(* CODESYS project VERSENY_25_F2

Project tree, tasks and I/O mapping:
  Device : CODESYS Control for PFC200 SL, 3S - Smart Software Solutions GmbH, version 4.1.0.0
    application Application
      libraries: Standard, 3.5.18.0 (System)
      task MainTask (cyclic, interval t#20ms, priority 1) calls PRG_TRIG, TESTPRG
      function BETWEEN [ST]
      CIMKEZO/
        data type ENUCIMKEZO
        function block FBCIMKEZO [ST]
      DOBOZ/
        data type ENUDOBOZ
        function block FBDOBOZ [ST]
      function block FBDOBOZ21212 [ST]
      global variables GVL
      global variables I
      LIFT/
        data type ENULIFT
        function block FBLIFT [ST]
      PALETTAZO/
        data type ENUPALETTAZO
        function block FBPALETTAZO [ST]
      program PLC_PRG [ST]
      PRESET/
        data type ENUPRESET
        function block FBPRESET [ST]
      program PRG_TRIG [ST]
      global variables Q
      RAKLAP/
        data type ENURAKLAP
        function block FBRAKLAP [ST]
      data type STATE
      program TESTPRG [ST]
      function block VILLOGO4 [ST]
    Pfc200Bus : Wago PFC200 internal bus, 3S - Smart Software Solutions GmbH, version 4.1.0.0
      _750_14xx_1 : 16DI, WAGO Kontakttechnik GmbH u. Co. KG, order no. 750-14xx, version 4.1.0.0
          unmapped channels: %IW10 Digital Inputs 0 - 15
      _750_14xx : 16DI, WAGO Kontakttechnik GmbH u. Co. KG, order no. 750-14xx, version 4.1.0.0
          unmapped channels: %IW5 Digital Inputs 0 - 15
      _750_15xx_1 : 16DO, WAGO Kontakttechnik GmbH u. Co. KG, order no. 750-15xx, version 4.1.0.0
          unmapped channels: %QW10 Digital Outputs 0 - 15
      _750_15xx : 16DO, WAGO Kontakttechnik GmbH u. Co. KG, order no. 750-15xx, version 4.1.0.0
          unmapped channels: %QW5 Digital Outputs 0 - 15
      _75x_459 : 75x-459/0..-000 4AI, 0-10 V, WAGO Kontakttechnik GmbH u. Co. KG, order no. 75x-459(/0..-000), version 4.1.0.0
          unmapped channels: Analog Input Channel 0, Analog Input Channel 1, Analog Input Channel 2, Analog Input Channel 3
      _75x_559 : 75x-559/0..-000 4AO, 0-10 V, WAGO Kontakttechnik GmbH u. Co. KG, order no. 75x-559(/0..-000), version 4.1.0.0
          unmapped channels: Analog Output Channel 0, Analog Output Channel 1, Analog Output Channel 2, Analog Output Channel 3
*)

// Device/Application/STATE
{attribute 'qualified_only'}
{attribute 'strict'}
TYPE STATE :
(
	enum_member := 0
);
END_TYPE

// Device/Application/CIMKEZO/ENUCIMKEZO
{attribute 'qualified_only'}
//{attribute 'strict'}
TYPE ENUCIMKEZO:
(
	PRESET := 0,
	CIMKEZZ := 1,
	DONE := 2
);
END_TYPE

// Device/Application/DOBOZ/ENUDOBOZ
{attribute 'qualified_only'}
//{attribute 'strict'}
TYPE ENUDOBOZ:
(
	PRESET := 0,
	CIKMEZO_CLEAR := 1,
	DONE := 2,
	GO := 3
);
END_TYPE

// Device/Application/LIFT/ENULIFT
{attribute 'qualified_only'}
//{attribute 'strict'}
TYPE ENULIFT:
(
	PRESET := 0,
	PARANCS_FEL := 1,
	PARANCS_LE := 2,
	LIFT_MOZOG := 3,
	DONE := 4
);
END_TYPE

// Device/Application/PALETTAZO/ENUPALETTAZO
{attribute 'qualified_only'}
//{attribute 'strict'}
TYPE ENUPALETTAZO:
(
	PRESET := 0,
	ELHALADT := 1,
	CELBA_ERT := 2,
	DOBOZOK_KESZ := 3,
	PALETTAZORA_TOVABBIT := 4,
	MEGERKEZETT := 5,
	BETOLO_VISSZA := 6,
	BETOLO_MEGY := 7,
	BETOLO_KESZ := 8,
	MEGFOG := 9,
	KINYIT := 10,
	DONE := 11
);
END_TYPE

// Device/Application/PRESET/ENUPRESET

{attribute 'qualified_only'}
//{attribute 'strict'}
TYPE ENUPRESET:
(
	PRESET := 0,
	MINDEN_LELAITAS := 1,
	LIFT_VISSZA := 2,
	DONE := 3
);
END_TYPE

// Device/Application/RAKLAP/ENURAKLAP
{attribute 'qualified_only'}
//{attribute 'strict'}
TYPE ENURAKLAP:
(
	PRESET := 0,
	WAIT := 1,
	DONE := 2,
	LEFELE := 3,
	LIFT_LE_VEGALAS := 4,
	LIFTBOL_KI := 5,
	LIFTBOL_KI_KETO := 6,
	GORGOS_MEHET := 7,
	BERAKO_INDIT := 8,
	LIFT_BEHORDO := 9,
	LIFT_FEL := 10,
	FELADAT_DONE := 11
);
END_TYPE

// Device/Application/GVL
{attribute 'qualified_only'}
VAR_GLOBAL
	STATE : STATE;
END_VAR

// Device/Application/I
{attribute 'qualified_only'}
VAR_GLOBAL
END_VAR

// Device/Application/Q
{attribute 'qualified_only'}
VAR_GLOBAL
END_VAR

// Device/Application/PRG_TRIG
PROGRAM PRG_TRIG
VAR
END_VAR

END_PROGRAM

// Device/Application/TESTPRG
PROGRAM TESTPRG
VAR
	LIFT : FBLIFT;
	FELFELE : BOOL;
	LEFELE : BOOL;
END_VAR

//LIFT TESZTELESE
IF I.I0 THEN
	FELFELE := TRUE;
	LEFELE := FALSE;
ELSIF I.I1 THEN
	LEFELE := TRUE;
	FELFELE := FALSE;
END_IF

LIFT(
	LEFELE:= LEFELE, 
	FELFELE:= FELFELE, 
	VEGALLASIG:= I.I2, 
	EN:= (I.I0 XOR I.I1), 
	DONE=> Q.Q0);

END_PROGRAM

// Device/Application/LIFT/FBLIFT
FUNCTION_BLOCK FBLIFT
VAR_INPUT
	LEFELE: BOOL;
	FELFELE: BOOL;
	VEGALLASIG: BOOL;
	EN: BOOL;
END_VAR
VAR_OUTPUT
	DONE: BOOL := FALSE;
END_VAR
VAR_IN_OUT
END_VAR
VAR
	LIFT: ENULIFT := ENULIFT.PRESET;
	VILLOGO4_PARANCS_VEGALLASIG_1_Q1: BOOL;
	BLANK_PARANCS_VEGALLASIG_1: BOOL;
	VILLOGO4_PARANCS_VEGALLASIG_1: VILLOGO4;
	TRANS_PARANCS_VEGALLASIG_PARANCS_FEL_T: TON;
	LELFELE: BOOL;
	TRANS_PARANCS_VEGALLASIG_PARANCS_LE_T: TON;
END_VAR

VILLOGO4_PARANCS_VEGALLASIG_1(T1:= T#1S, T2:= T#1S, T3:= T#0S, T4:= T#0S, Q1:= VILLOGO4_PARANCS_VEGALLASIG_1_Q1, Q2:= BLANK_PARANCS_VEGALLASIG_1, Q3:= BLANK_PARANCS_VEGALLASIG_1, Q4:= BLANK_PARANCS_VEGALLASIG_1, EN:= (LIFT = ENULIFT.PARANCS_VEGALLASIG));
TRANS_PARANCS_VEGALLASIG_PARANCS_FEL_T(PT:= T#5S, IN:= FELFELE AND (LIFT = ENULIFT.PARANCS_VEGALLASIG));
TRANS_PARANCS_VEGALLASIG_PARANCS_LE_T(PT:= T#5S, IN:= LELFELE AND (LIFT = ENULIFT.PARANCS_VEGALLASIG));

IF NOT EN THEN
	LIFT := ENULIFT.PRESET;
	LELFELE := FALSE;
	BLANK_PARANCS_VEGALLASIG_1 := FALSE;
	VILLOGO4_PARANCS_VEGALLASIG_1_Q1 := FALSE;
	DONE := FALSE;
	RETURN;
END_IF


CASE LIFT OF
	ENULIFT.PRESET:
	Q.LIFT_VEGALLASIG := VEGALLASIG;

	IF FELFELE AND NOT VEGALLASIG THEN
		LIFT := ENULIFT.PARANCS_FEL;
	ELSIF LEFELE AND NOT VEGALLASIG THEN
		LIFT := ENULIFT.PARANCS_LE;
	ELSIF VEGALLASIG AND (FELFELE OR LEFELE) THEN
		LIFT := ENULIFT.PARANCS_VEGALLASIG;
	END_IF

	ENULIFT.PARANCS_FEL:
	Q.LIFT_FEL := TRUE;

	IF I.LIFT_MOZOG THEN
		LIFT := ENULIFT.LIFT_MOZOG;
	END_IF

	ENULIFT.PARANCS_LE:
	Q.LIFT_LE := TRUE;

	IF I.LIFT_MOZOG THEN
		LIFT := ENULIFT.LIFT_MOZOG;
	END_IF


	ENULIFT.LIFT_MOZOG:
	IF NOT (VEGALLASIG AND NOT I.I15) THEN
		Q.LIFT_FEL := FALSE;
		Q.LIFT_LE := FALSE;
		Q.LIFT_VEGALLASIG := FALSE;
	END_IF

	IF GVL.LIFT_MOZOG_F_TRIG.Q THEN
		Q.LIFT_FEL := FALSE;
		Q.LIFT_LE := FALSE;
		Q.LIFT_VEGALLASIG := FALSE;
		

		LIFT := ENULIFT.DONE;
	END_IF



	ENULIFT.PARANCS_VEGALLASIG:

	IF TRANS_PARANCS_VEGALLASIG_PARANCS_FEL_T.Q THEN
		LIFT := ENULIFT.PARANCS_FEL;
	ELSIF TRANS_PARANCS_VEGALLASIG_PARANCS_LE_T.Q THEN
		LIFT := ENULIFT.PARANCS_LE;
	END_IF

END_CASE

DONE := (LIFT = ENULIFT.DONE);
Q.HORN := (VILLOGO4_PARANCS_VEGALLASIG_1_Q1 AND (LIFT = ENULIFT.PARANCS_VEGALLASIG));

END_FUNCTION_BLOCK

// Device/Application/VILLOGO4
FUNCTION_BLOCK VILLOGO4
VAR_INPUT
	T1: TIME;
	T2: TIME;
	T3: TIME;
	T4: TIME;
END_VAR
VAR_IN_OUT
	Q1: BOOL;
	Q2: BOOL;
	Q3: BOOL;
	Q4: BOOL;
END_VAR
VAR
	T1_TON: TON;
	T2_TON: TON;
	T3_TON: TON;
	T4_TON: TON;
END_VAR
VAR_INPUT
	EN: BOOL := FALSE;
END_VAR
VAR
	EN_F_TRIG: F_TRIG;
	EN_R_TRIG: R_TRIG;
	STATE: INT := 0;
	PREV_STATE: INT := 0;
END_VAR

EN_F_TRIG(CLK := EN);
EN_R_TRIG(CLK := EN);

IF EN_F_TRIG.Q THEN
	Q1 := FALSE;
	Q2 := FALSE;
	Q3 := FALSE;
	Q4 := FALSE;
	T1_TON.PT := T1_TON.ET;
	T2_TON.PT := T2_TON.ET;
	T3_TON.PT := T3_TON.ET;
	T4_TON.PT := T4_TON.ET;
	STATE := 0;
ELSIF EN_R_TRIG.Q THEN
		Q1 := TRUE;
END_IF

IF NOT EN THEN
	RETURN;
END_IF

T1_TON(IN:= EN_R_TRIG.Q OR (STATE = 0), PT:= T1);
T2_TON(IN:= STATE = 1, PT:= T2);
T3_TON(IN:= STATE = 2, PT:= T3);
T4_TON(IN:= STATE = 3, PT:= T4);

IF T1_TON.Q THEN
	Q1 := FALSE;
	Q2 := TRUE;
END_IF
IF T2_TON.Q THEN
	Q2 := FALSE;
	Q3 := TRUE;
END_IF
IF T3_TON.Q THEN
	Q3 := FALSE;
	Q4 := TRUE;
END_IF
IF T4_TON.Q THEN
	Q4 := FALSE;
	Q1 := TRUE;
END_IF

IF T1_TON.Q OR T2_TON.Q OR T3_TON.Q OR T4_TON.Q THEN
	STATE := STATE + 1;
END_IF

IF STATE > 3 THEN
	STATE := 0;
END_IF

END_FUNCTION_BLOCK

// Device/Application/BETWEEN
FUNCTION BETWEEN : BOOL
VAR_INPUT
	STATE : INT;
	LOW : INT;
	HIGH : INT;
END_VAR
VAR_OUTPUT
END_VAR
VAR
	EN_TRIG : F_TRIG;
END_VAR

IF STATE >= LOW AND STATE <= HIGH THEN
	BETWEEN := TRUE;
ELSE 
	BETWEEN := FALSE;
END_IF

END_FUNCTION

// Device/Application/FBDOBOZ21212
FUNCTION_BLOCK FBDOBOZ21212
VAR_INPUT
	EN : BOOL;
END_VAR
VAR_OUTPUT
	DONE : BOOL;
END_VAR
VAR
END_VAR

END_FUNCTION_BLOCK

// Device/Application/PLC_PRG
PROGRAM PLC_PRG
VAR
END_VAR

%QW10 := %IW10;

END_PROGRAM

// Device/Application/CIMKEZO/FBCIMKEZO
FUNCTION_BLOCK FBCIMKEZO
VAR_INPUT
	EN: BOOL;
END_VAR
VAR_OUTPUT
	DONE: BOOL := FALSE;
END_VAR
VAR_IN_OUT
END_VAR
VAR
	CIMKEZO: ENUCIMKEZO := ENUCIMKEZO.PRESET;
	TRANS_CIMKEZZ_DONE_T: TON;
END_VAR

TRANS_CIMKEZZ_DONE_T(PT:= GVL.CIMKEZO_TIME, IN:= (CIMKEZO = ENUCIMKEZO.CIMKEZZ));

IF NOT EN THEN
	CIMKEZO := ENUCIMKEZO.PRESET;
	DONE := FALSE;
	RETURN;
END_IF


CASE CIMKEZO OF

	ENUCIMKEZO.PRESET:

	IF GVL.DOBOZ_CIMKEZONEL_F_TRIG.Q THEN
		CIMKEZO := ENUCIMKEZO.CIMKEZZ;
	END_IF


	ENUCIMKEZO.CIMKEZZ:

	IF TRANS_CIMKEZZ_DONE_T.Q THEN
		CIMKEZO := ENUCIMKEZO.DONE;
	END_IF


	ENUCIMKEZO.DONE:

	IF TRUE THEN
		CIMKEZO := ENUCIMKEZO.PRESET;
	END_IF

END_CASE

DONE := (CIMKEZO = ENUCIMKEZO.DONE);
Q.CIMKEZO := (CIMKEZO = ENUCIMKEZO.CIMKEZZ);

END_FUNCTION_BLOCK

// Device/Application/DOBOZ/FBDOBOZ
FUNCTION_BLOCK FBDOBOZ
VAR_INPUT
	MODE: BOOL;
	EN: BOOL;
END_VAR
VAR_OUTPUT
	DONE: BOOL := FALSE;
END_VAR
VAR_IN_OUT
END_VAR
VAR
	DOBOZ: ENUDOBOZ := ENUDOBOZ.PRESET;
	CIMKEZO: FBCIMKEZO;
	PALETTAZO: FBPALETTAZO;
	MAX_DOBOZ: INT;
	MAX_OSZLOP: INT;
END_VAR

PALETTAZO(MAX_DOBOZ := MAX_DOBOZ, MAX_OSZLOP := MAX_OSZLOP, EN:= (DOBOZ = ENUDOBOZ.CIKMEZO_CLEAR) OR (DOBOZ = ENUDOBOZ.GO));
CIMKEZO(EN:= (DOBOZ = ENUDOBOZ.GO));

IF NOT EN THEN
	DOBOZ := ENUDOBOZ.PRESET;
	MAX_OSZLOP := 0;
	MAX_DOBOZ := 0;
	DONE := FALSE;
	RETURN;
END_IF


CASE DOBOZ OF

	ENUDOBOZ.PRESET:

	IF TRUE THEN
		DOBOZ := ENUDOBOZ.GO;
	END_IF


	ENUDOBOZ.CIKMEZO_CLEAR:

	IF TRUE THEN
		DOBOZ := ENUDOBOZ.GO;
	END_IF



	ENUDOBOZ.GO:
	IF MODE THEN
		Q.TERELO := TRUE;
		MAX_DOBOZ := 3;
		MAX_OSZLOP := 2;
	ELSE
		Q.TERELO := FALSE;
		MAX_DOBOZ := 2;
		MAX_OSZLOP := 3;
	END_IF

	IF CIMKEZO.DONE THEN
		DOBOZ := ENUDOBOZ.CIKMEZO_CLEAR;
	ELSIF PALETTAZO.DONE THEN
		DOBOZ := ENUDOBOZ.DONE;
	END_IF

END_CASE

DONE := (DOBOZ = ENUDOBOZ.DONE);

END_FUNCTION_BLOCK

// Device/Application/PALETTAZO/FBPALETTAZO
FUNCTION_BLOCK FBPALETTAZO
VAR_INPUT
	MAX_DOBOZ: INT;
	MAX_OSZLOP: INT;
	EN: BOOL;
END_VAR
VAR_OUTPUT
	ATHALADT_DOBOZOK: INT;
	KESZ_OSZLOPOK: INT;
	DONE: BOOL := FALSE;
END_VAR
VAR_IN_OUT
END_VAR
VAR
	PALETTAZO: ENUPALETTAZO := ENUPALETTAZO.PRESET;
	TRANS_ELHALADT_CELBA_ERT_T: TON;
	ATHALADT_DOBOZOK_SZAMA: INT;
END_VAR

TRANS_ELHALADT_CELBA_ERT_T(PT:= GVL.CELBA_ER_TIME, IN:= (PALETTAZO = ENUPALETTAZO.ELHALADT));

IF NOT EN THEN
	PALETTAZO := ENUPALETTAZO.PRESET;
	ATHALADT_DOBOZOK_SZAMA := 0;
	DONE := FALSE;
	KESZ_OSZLOPOK := 0;
	ATHALADT_DOBOZOK := 0;
	RETURN;
END_IF


CASE PALETTAZO OF
	ENUPALETTAZO.PRESET:
	Q.BEHORDO := TRUE;
	Q.PALETTAZO_OPEN := FALSE;

	IF GVL.BEHORDO_Z1_R_TRIG.Q THEN
		PALETTAZO := ENUPALETTAZO.MEGERKEZETT;
	END_IF


	ENUPALETTAZO.ELHALADT:

	IF TRANS_ELHALADT_CELBA_ERT_T.Q THEN
		ATHALADT_DOBOZOK_SZAMA := ATHALADT_DOBOZOK_SZAMA + 1;

		PALETTAZO := ENUPALETTAZO.CELBA_ERT;
	END_IF


	ENUPALETTAZO.CELBA_ERT:

	IF ATHALADT_DOBOZOK_SZAMA < MAX_DOBOZ THEN
		PALETTAZO := ENUPALETTAZO.PRESET;
	ELSIF ATHALADT_DOBOZOK_SZAMA = MAX_DOBOZ THEN
		PALETTAZO := ENUPALETTAZO.DOBOZOK_KESZ;
	END_IF

	ENUPALETTAZO.DOBOZOK_KESZ:
	Q.BEHORDO := FALSE;
	Q.PALETTAZO_SZALAG := FALSE;

	IF I.PALETTAZO_CLOSED AND I.PALETTAZO_BETOLO_VEGALLAS AND I.PALETTAZO_DOBOZ_MEGFOGVA AND NOT Q.PALETTAZO_BETOLO AND NOT Q.PALETTAZO_MEGFOGO THEN
		PALETTAZO := ENUPALETTAZO.PALETTAZORA_TOVABBIT;
	END_IF


	ENUPALETTAZO.PALETTAZORA_TOVABBIT:

	IF GVL.PALETTAZO_BETOLO_VEGALLAS_R_TRIG.Q THEN
		PALETTAZO := ENUPALETTAZO.BETOLO_VISSZA;
	END_IF

	ENUPALETTAZO.MEGERKEZETT:
	Q.PALETTAZO_SZALAG := TRUE;

	IF GVL.BEHORDO_Z1_F_TRIG.Q THEN
		PALETTAZO := ENUPALETTAZO.ELHALADT;
	END_IF


	ENUPALETTAZO.BETOLO_VISSZA:

	IF GVL.PALETTAZO_BETOLO_VEGALLAS_F_TRIG.Q THEN
		PALETTAZO := ENUPALETTAZO.BETOLO_MEGY;
	END_IF


	ENUPALETTAZO.BETOLO_MEGY:

	IF GVL.PALETTAZO_BETOLO_VEGALLAS_R_TRIG.Q THEN
		KESZ_OSZLOPOK := KESZ_OSZLOPOK + 1;

		PALETTAZO := ENUPALETTAZO.BETOLO_KESZ;
	END_IF


	ENUPALETTAZO.BETOLO_KESZ:

	IF KESZ_OSZLOPOK < MAX_OSZLOP THEN
		PALETTAZO := ENUPALETTAZO.PRESET;
	ELSIF KESZ_OSZLOPOK = MAX_OSZLOP THEN
		PALETTAZO := ENUPALETTAZO.MEGFOG;
	END_IF


	ENUPALETTAZO.MEGFOG:

	IF GVL.PALETTAZO_DOBOZ_MEGFOGVA_R_TRIG.Q AND NOT I.LIFT_MOZOG THEN
		PALETTAZO := ENUPALETTAZO.KINYIT;
	END_IF

	ENUPALETTAZO.KINYIT:
	Q.PALETTAZO_OPEN := TRUE;

	IF TRUE THEN
		PALETTAZO := ENUPALETTAZO.DONE;
	END_IF


END_CASE

DONE := (PALETTAZO = ENUPALETTAZO.DONE);
Q.PALETTAZO_BETOLO := (PALETTAZO = ENUPALETTAZO.PALETTAZORA_TOVABBIT);
Q.PALETTAZO_MEGFOGO := (PALETTAZO = ENUPALETTAZO.MEGFOG);

END_FUNCTION_BLOCK

// Device/Application/PRESET/FBPRESET
FUNCTION_BLOCK FBPRESET
VAR_INPUT
	EN: BOOL;
END_VAR
VAR_OUTPUT
	DONE: BOOL := FALSE;
END_VAR
VAR_IN_OUT
END_VAR
VAR
	PRESET: ENUPRESET := ENUPRESET.PRESET;
END_VAR

IF NOT EN THEN
	PRESET := ENUPRESET.PRESET;
	DONE := FALSE;
	RETURN;
END_IF


CASE PRESET OF

	ENUPRESET.PRESET:

	IF EN THEN
		PRESET := ENUPRESET.MINDEN_LELAITAS;
	END_IF


	ENUPRESET.MINDEN_LELAITAS:
	%QW10 := 0;

	IF TRUE THEN
		PRESET := ENUPRESET.LIFT_VISSZA;
	END_IF


	ENUPRESET.LIFT_VISSZA:

	IF GVL.LIFT_MOZOG_F_TRIG.Q OR GVL.LIFT_LENT THEN
		PRESET := ENUPRESET.DONE;
	END_IF


END_CASE

DONE := (PRESET = ENUPRESET.DONE);
Q.LIFT_LE := (PRESET = ENUPRESET.LIFT_VISSZA);

END_FUNCTION_BLOCK

// Device/Application/RAKLAP/FBRAKLAP
FUNCTION_BLOCK FBRAKLAP
VAR_INPUT
	LEFELE: BOOL;
	KIRAKAS: BOOL;
	BERAKAS: BOOL;
	HARMADIK: BOOL;
	STOP: BOOL;
	EN: BOOL;
END_VAR
VAR_OUTPUT
	FELADAT_DONE: BOOL;
	DONE: BOOL := FALSE;
END_VAR
VAR_IN_OUT
END_VAR
VAR
	RAKLAP: ENURAKLAP := ENURAKLAP.PRESET;
	LIFT: FBLIFT;
	LEFELE_MENJ: BOOL;
	FELFELE_MENJ: BOOL;
	VEGALAS_MENJ: BOOL;
	LIFT_BEHORDO: BOOL;
	TRANS_GORGOS_MEHET_DONE_T: TON;
	IDOMENTES : TIME;
END_VAR

LIFT(EN:= (RAKLAP = ENURAKLAP.LEFELE) OR 
		  (RAKLAP = ENURAKLAP.LIFT_FEL) OR 
          (RAKLAP = ENURAKLAP.LIFT_LE_VEGALAS) );
TRANS_GORGOS_MEHET_DONE_T(PT:= T#3S, IN:= ((RAKLAP = ENURAKLAP.GORGOS_MEHET) AND (NOT STOP)) );

LIFT.FELFELE := FELFELE_MENJ;
LIFT.LEFELE := LEFELE_MENJ;
LIFT.VEGALLASIG := VEGALAS_MENJ;


IF NOT EN THEN
	RAKLAP := ENURAKLAP.PRESET;
	LIFT_BEHORDO := FALSE;
	VEGALAS_MENJ := FALSE;
	FELFELE_MENJ := FALSE;
	LEFELE_MENJ := FALSE;
	DONE := FALSE;
	FELADAT_DONE := FALSE;
	RETURN;
END_IF


CASE RAKLAP OF

	ENURAKLAP.PRESET:

	IF EN THEN
		RAKLAP := ENURAKLAP.WAIT;
	END_IF


	ENURAKLAP.WAIT:

	IF LEFELE AND (NOT STOP )THEN
		RAKLAP := ENURAKLAP.LEFELE;
	ELSIF KIRAKAS  AND (NOT STOP ) THEN
		RAKLAP := ENURAKLAP.LIFT_LE_VEGALAS;
	ELSIF BERAKAS AND (NOT STOP ) THEN
		RAKLAP := ENURAKLAP.BERAKO_INDIT;
	END_IF



	ENURAKLAP.LEFELE:

	IF LIFT.DONE AND (NOT STOP ) THEN
		RAKLAP := ENURAKLAP.DONE;
	END_IF


	ENURAKLAP.LIFT_LE_VEGALAS:

	IF LIFT.DONE AND (NOT STOP ) THEN
		RAKLAP := ENURAKLAP.LIFTBOL_KI;
	END_IF


	ENURAKLAP.LIFTBOL_KI:

	IF (NOT I.LIFT_PALETTA_BACK_1) AND (NOT STOP ) THEN
		RAKLAP := ENURAKLAP.LIFTBOL_KI_KETO;
	END_IF


	ENURAKLAP.LIFTBOL_KI_KETO:

	IF (NOT I.LIFT_PALETTA_FRONT_2) AND (NOT STOP )  THEN
		RAKLAP := ENURAKLAP.GORGOS_MEHET;
	END_IF


	ENURAKLAP.GORGOS_MEHET:

	IF TRANS_GORGOS_MEHET_DONE_T.Q THEN
		RAKLAP := ENURAKLAP.DONE;
	ELSIF I.GORGOS_PALYA_Z1 AND HARMADIK AND (NOT STOP ) THEN
		RAKLAP := ENURAKLAP.FELADAT_DONE;
	END_IF


	ENURAKLAP.BERAKO_INDIT:

	IF I.LIFT_PALETTA_BACK_1 AND (NOT STOP ) THEN
		RAKLAP := ENURAKLAP.LIFT_BEHORDO;
	END_IF


	ENURAKLAP.LIFT_BEHORDO:

	IF I.LIFT_PALETTA_FRONT_2 AND (NOT STOP ) THEN
		RAKLAP := ENURAKLAP.LIFT_FEL;
	END_IF


	ENURAKLAP.LIFT_FEL:

	IF LIFT.DONE THEN
		RAKLAP := ENURAKLAP.DONE;
	END_IF


END_CASE

DONE := (RAKLAP = ENURAKLAP.DONE) OR (RAKLAP = ENURAKLAP.FELADAT_DONE);
FELFELE_MENJ := (RAKLAP = ENURAKLAP.LIFT_FEL) AND (NOT STOP ) ;
LEFELE_MENJ := (RAKLAP = ENURAKLAP.LEFELE) OR (RAKLAP = ENURAKLAP.LIFT_LE_VEGALAS) AND (NOT STOP ) ;
LIFT_BEHORDO := (RAKLAP = ENURAKLAP.LIFT_BEHORDO) AND (NOT STOP ) ;
Q.GORGOS_PALYA := (RAKLAP = ENURAKLAP.BERAKO_INDIT) OR (RAKLAP = ENURAKLAP.LIFT_BEHORDO) AND (NOT STOP );
Q.KIHORDO := (RAKLAP = ENURAKLAP.GORGOS_MEHET) OR (RAKLAP = ENURAKLAP.LIFTBOL_KI_KETO) AND (NOT STOP ) ;
Q.LIFT_BEHORDO := (RAKLAP = ENURAKLAP.LIFTBOL_KI) OR (RAKLAP = ENURAKLAP.LIFTBOL_KI_KETO) AND (NOT STOP );
VEGALAS_MENJ := (RAKLAP = ENURAKLAP.LIFT_FEL) OR (RAKLAP = ENURAKLAP.LIFT_LE_VEGALAS) AND (NOT STOP );

END_FUNCTION_BLOCK
